// TIA Portal project "Cm19_431 2019_11_11" (V15.1)

(* hardware
DEVICE "ET 200SP station_1"  ET 200SP-Station
   slot 0: "Telaio di montaggio_0"  Rack  6ES5 710-8MAx1
   slot 1: "PLC_1"  CPU 1510SP-1 PN  6ES7 510-1DJ01-0AB0  V2.6
   slot 2: "DI 16x24VDC ST_1"  DI 16x24VDC ST  6ES7 131-6BH01-0BA0  V0.0
      slot 1: "DI 16x24VDC ST_1"  DI 16x24VDC ST
   slot 3: "DQ 16x24VDC/0.5A ST_1"  DQ 16x24VDC/0.5A ST  6ES7 132-6BH01-0BA0  V0.0
      slot 1: "DQ 16x24VDC/0.5A ST_1"  DQ 16x24VDC/0.5A ST
   slot 4: "Modulo server_1"  Server module  6ES7 193-6PA00-0AA0  V1.1
      slot 1: "Modulo server_1"  Server module
   slot 127: "BA 2xRJ45"  BA 2xRJ45  6ES7 193-6AR00-0AA0  V0.0
      slot 32769: "Port_1"  6ES7 193-6AR00-0AA0
      slot 32770: "Port_2"  6ES7 193-6AR00-0AA0
DEVICE "HMI_1"  KTP700F Mobile
   slot 0: "HMI_1"  KTP700F Mobile  6AV2 125-2GB23-0AX0  15.1.0.0
   slot 1: "HMI_RT_1"  KTP700F Mobile  6AV2 125-2GB23-0AX0  15.1.0.0
   slot 5: "HMI_1.IE_CP_1"  PROFINET Interface  15.0.1.0
      slot 1: "Interfaccia_1 PROFINET"  PROFINET Interface
         slot 1: "Porta_1"  Port
DEVICE "GSD device_1"  GSD.Device.PN
   slot 0: "Telaio di montaggio"  Rack  V1.0
   slot 0: "CPX"  CPX Rev 30  TN 197330  V4.2.30
      slot 0: "CPX Rev 30"  CPX Rev 30
      slot 1: "PN-IO Interface"  PN-IO Interface
         slot 1: "Port 1"  Port 1
         slot 2: "Port 2"  Port 2
   slot 1: "FB33 PNIO Module_1"  FB33 PNIO Module  TN 548755, CPX-FB33, Code F33
      slot 0: "FB33 PNIO Module"  FB33 PNIO Module
DEVICE "GSD device_2"  GSD.Device.PN
   slot 0: "Telaio di montaggio"  Rack  V1.0
   slot 0: "AP-I-PN"  CPX-AP-I V1  CPX-AP-I  V1.0.0
      slot 0: "CPX-AP-I V1"  CPX-AP-I V1
      slot 1: "CPX-AP-I-PN-M12_1"  CPX-AP-I-PN-M12  8086607
         slot 0: "CPX-AP-I-PN-M12"  CPX-AP-I-PN-M12  8086607
      slot 1: "PN-IO Interface"  PN-IO Interface
         slot 1: "Port 1"  Port 1
         slot 2: "Port 2"  Port 2
*)

// ===== PLC "PLC_1"  CPU 1510SP-1 PN =====

VAR_GLOBAL   // PLC tag table "Merker"
   "CICLO ST.9" AT %M80.0 : Bool;   // CICLO ST.9
   "CICLO ST.10" AT %M80.1 : Bool;   // CICLO ST.10
   "CICLI STAZIONI" AT %MW80 : Word;   // CICLI STAZIONI
   "CICLO GENERALE" AT %M70.0 : Bool;   // FLAG DI CICLO GENERALE
   "RICHIESTA ARRESTO A FINE CICLO" AT %M18.1 : Bool;   // RICHIESTA ARRESTO A FINE CICLO
   "MACCHINA IN FINE CICLO" AT %M18.3 : Bool;   // MACCHINA IN FINE CICLO
   "ALLARMI SISTEMA" AT %MB20 : Byte;   // ALLARMI SISTEMA
   "CICLO ST.11" AT %M80.2 : Bool;   // CICLO ST.11
   "CICLO ST.12" AT %M80.3 : Bool;   // CICLO ST.12
   "CICLO ST.13" AT %M80.4 : Bool;   // CICLO ST.13
   "CICLO ST.14" AT %M80.5 : Bool;   // CICLO ST.14
   "CICLO ST.15" AT %M80.6 : Bool;   // CICLO ST.15
   "CICLO ST.16" AT %M80.7 : Bool;   // CICLO ST.16
   "CICLO ST.1" AT %M81.0 : Bool;   // CICLO ST.1
   "CICLO ST.2" AT %M81.1 : Bool;   // CICLO ST.2
   "CICLO ST.3" AT %M81.2 : Bool;   // CICLO ST.3
   "CICLO ST.4" AT %M81.3 : Bool;   // CICLO ST.4
   "CICLO ST.5" AT %M81.4 : Bool;   // CICLO ST.5
   "CICLO ST.6" AT %M81.5 : Bool;   // CICLO ST.6
   "CICLO ST.7" AT %M81.6 : Bool;   // CICLO ST.7
   "CICLO ST.8" AT %M81.7 : Bool;   // CICLO ST.8
   "PUL. CICLO RILASCIATO" AT %M70.1 : Bool;   // PULSANTE DI CICLO RILASCIATO
   "STAZIONI PRESENTI" AT %MW6 : Word;   // STAZIONI PRESENTI
   "STAZIONI INCLUSE" AT %MW8 : Word;   // STAZIONI INCLUSE
   "St.9 PRESENTE" AT %M6.0 : Bool;   // St.9 PRESENTE
   "St.10 PRESENTE" AT %M6.1 : Bool;   // St.10 PRESENTE
   "St.11 PRESENTE" AT %M6.2 : Bool;   // St.11 PRESENTE
   "St.12 PRESENTE" AT %M6.3 : Bool;   // St.12 PRESENTE
   "St.13 PRESENTE" AT %M6.4 : Bool;   // St.13 PRESENTE
   "St.14 PRESENTE" AT %M6.5 : Bool;   // St.14 PRESENTE
   "St.15 PRESENTE" AT %M6.6 : Bool;   // St.15 PRESENTE
   "St.16 PRESENTE" AT %M6.7 : Bool;   // St.16 PRESENTE
   "St.1 PRESENTE" AT %M7.0 : Bool;   // St.1 PRESENTE
   "St.2 PRESENTE" AT %M7.1 : Bool;   // St.2 PRESENTE
   "St.3 PRESENTE" AT %M7.2 : Bool;   // St.3 PRESENTE
   "St.4 PRESENTE" AT %M7.3 : Bool;   // St.4 PRESENTE
   "St.5 PRESENTE" AT %M7.4 : Bool;   // St.5 PRESENTE
   "St.6 PRESENTE" AT %M7.5 : Bool;   // St.6 PRESENTE
   "St.7 PRESENTE" AT %M7.6 : Bool;   // St.7 PRESENTE
   "St.8 PRESENTE" AT %M7.7 : Bool;   // St.8 PRESENTE
   "ST.9 INCLUSA" AT %M8.0 : Bool;   // ST.9 INCLUSA
   "ST.10 INCLUSA" AT %M8.1 : Bool;   // ST.10 INCLUSA
   "ST.11 INCLUSA" AT %M8.2 : Bool;   // ST.11 INCLUSA
   "ST.12 INCLUSA" AT %M8.3 : Bool;   // ST.12 INCLUSA
   "ST.13 INCLUSA" AT %M8.4 : Bool;   // ST.13 INCLUSA
   "ST.14 INCLUSA" AT %M8.5 : Bool;   // ST.14 INCLUSA
   "ST.15 INCLUSA" AT %M8.6 : Bool;   // ST.15 INCLUSA
   "ST.16 INCLUSA" AT %M8.7 : Bool;   // ST.16 INCLUSA
   "ST.1 INCLUSA" AT %M9.0 : Bool;   // ST.1 INCLUSA
   "ST.2 INCLUSA" AT %M9.1 : Bool;   // ST.2 INCLUSA
   "ST.3 INCLUSA" AT %M9.2 : Bool;   // ST.3 INCLUSA
   "ST.4 INCLUSA" AT %M9.3 : Bool;   // ST.4 INCLUSA
   "ST.5 INCLUSA" AT %M9.4 : Bool;   // ST.5 INCLUSA
   "ST.6 INCLUSA" AT %M9.5 : Bool;   // ST.6 INCLUSA
   "ST.7 INCLUSA" AT %M9.6 : Bool;   // ST.7 INCLUSA
   "ST.8 INCLUSA" AT %M9.7 : Bool;   // ST.8 INCLUSA
END_VAR

VAR_GLOBAL   // PLC tag table "Output"
   "LAMPADA CICLO" AT %A0.0 : Bool;
   "LAMPADE ALLARME" AT %A0.1 : Bool;
   "LAMPADA VIB. VUOTI" AT %A0.2 : Bool;
   "LAMPADA ARR.FINE CICLO" AT %A0.3 : Bool;
   "LAMPADA MANUALE" AT %A0.4 : Bool;
   "MOTORE ROTAZIONE TAVOLA" AT %A0.5 : Bool;
   "MOTORE NASTRO TRASPORTATORE ST.1" AT %A0.6 : Bool;
   "A0.7" AT %A0.7 : Bool;
   "A1.0" AT %A1.0 : Bool;
   "A1.1" AT %A1.1 : Bool;
   "A1.2" AT %A1.2 : Bool;
   "A1.3" AT %A1.3 : Bool;
   "A1.4" AT %A1.4 : Bool;
   "A1.5" AT %A1.5 : Bool;
   "A1.6" AT %A1.6 : Bool;
   "A1.7" AT %A1.7 : Bool;
END_VAR

VAR_GLOBAL   // PLC tag table "Input"
   "PULSANTI CICLO" AT %E0.1 : Bool;
   "POTENZA INSERITA" AT %E0.0 : Bool;
   "PULSANTI TACITAZIONE ALLARMI" AT %E0.2 : Bool;
   "SEL.SVUOTAMENTO TAVOLA" AT %E0.3 : Bool;
   "SEL.SINGOLO CONTINUO" AT %E0.4 : Bool;
   "TERMICI OK" AT %E0.5 : Bool;
   "SICUREZZA PARATIE" AT %E0.6 : Bool;
   "PULSANTE UOMO MORTO TASTIERINO" AT %E0.7 : Bool;
   "E1.0" AT %E1.0 : Bool;
   "E1.1" AT %E1.1 : Bool;
   "E1.2" AT %E1.2 : Bool;
   "E1.3" AT %E1.3 : Bool;
   "E1.4" AT %E1.4 : Bool;
   "E1.5" AT %E1.5 : Bool;
   "E1.6" AT %E1.6 : Bool;
   "E1.7" AT %E1.7 : Bool;
END_VAR

FUNCTION "FC1 CICLO GENERALE" : Void   // FC1, LAD
TITLE = GESTIONE CICLO GENERALE
{ S7_Optimized_Access := 'TRUE' }
VERSION : 0.1
BEGIN

REGION Network 1 (STL): FLAG DI CICLO GENERALE
         L     "CICLI STAZIONI";  // Verifica che tutte le stazioni siano a fine ciclo
         L     0;
         ==I;
         R     "CICLO GENERALE";
         R     "RICHIESTA ARRESTO A FINE CICLO";
         S     "MACCHINA IN FINE CICLO";

         A(;  // Allarmi presenti
         L     "ALLARMI SISTEMA";
         L     0;
         <>I;
         );
         JC    M001;

         A     "PULSANTI CICLO";  // Pulsante CICLO
         JC    M004;
         S     "PUL. CICLO RILASCIATO";
         BEU;

   M004: A     "PUL. CICLO RILASCIATO";  // Memoria puls. ciclo rilasciato
         JC    M002;
         BEU;

   M002: AN    "CICLO GENERALE";  // Maccina in ciclo
         JC    M003;
         S     "RICHIESTA ARRESTO A FINE CICLO";  // Setta arresto a fine ciclo
         R     "PUL. CICLO RILASCIATO";
         JU    M001;

   M003: S     "CICLO GENERALE";
         L     "STAZIONI PRESENTI";  // Stazioni presenti
         L     "STAZIONI INCLUSE";  // Stazioni incluse
         AW;
         T     "CICLI STAZIONI";  // Setta ciclo alle stazioni
         R     "PUL. CICLO RILASCIATO";
         R     "RICHIESTA ARRESTO A FINE CICLO";
         R     "MACCHINA IN FINE CICLO";
   M001: BE;
END_REGION
END_FUNCTION

ORGANIZATION_BLOCK "Main"   // OB1, LAD, ProgramCycle
TITLE = "Main Program Sweep (Cycle)"
{ S7_Optimized_Access := 'TRUE' }
VERSION : 0.1
   VAR_INPUT
      Initial_Call : Bool;   // Initial call of this OB
      Remanence : Bool;   // =True, if remanent data are available
   END_VAR
BEGIN
END_ORGANIZATION_BLOCK

(* ===== HMI "HMI_RT_1" =====
system functions are stored by id; their names below are inferred from use
connection "HMI_Collegamento_1": ETHERNET, S7_1500_OMS

HMI tags "Tabella delle variabili standard"
   "Variabile_Numero di pagina" : UInt, internal

text list "Elenco testi_Nome della pagina": 1 'Pagina base'

screen "Pagina base" 800x408, template "Modello_1"
   on GenerateScreen: SetTag("Variabile_Numero di pagina", 1)
   TextField "HmiScreenItemData" at 80,153 size 640x25; Text 'Benvenuto in HMI_1 (KTP700F Mobile)!'

Template "Modello_1" 800x408
   Button "Esci" at 727,335 size 71x71; TextOff 'Esci'; PictureOff "ExitRuntime_KTP700F_Mobile_TR"; PictureOn "ExitRuntime_KTP700F_Mobile_TR"
      on Release: StopRuntime(0)
   Button "Template_Button" at 654,335 size 71x71; TextOff 'Text'
   Button "Template_Button_1" at 582,335 size 71x71; TextOff 'Text'
   Button "Template_Button_2" at 509,335 size 71x71; TextOff 'Text'
   Button "Template_Button_3" at 437,335 size 71x71; TextOff 'Text'
   Button "Template_Button_4" at 364,335 size 71x71; TextOff 'Text'
   Button "Template_Button_5" at 291,335 size 71x71; TextOff 'Text'
   Button "Template_Button_6" at 219,335 size 71x71; TextOff 'Text'
   Button "Template_Button_7" at 146,335 size 71x71; TextOff 'Text'
   Button "Segnalazioni" at 74,335 size 71x71; TextOff 'Segnalazioni'; PictureOff "AlarmDisplay_KTP700F_Mobile_TR"; PictureOn "AlarmDisplay_KTP700F_Mobile_TR"
      on Release: function_ef3f5d25("Finestra delle segnalazioni_Non riconosciuta", -1)
   Button "Pagina iniziale" at 1,335 size 71x71; TextOff 'Pagina iniziale'; PictureOff "NavigateHome_KTP700F_Mobile_TR"; PictureOn "NavigateHome_KTP700F_Mobile_TR"
      on Release: ActivateScreen("Pagina base", 0)
*)